// SIMATIC S7-200 project (STEP 7-Micro/WIN), CPU 221 REL 01.10

ORGANIZATION_BLOCK 主程序:OB1
TITLE=程序注释
BEGIN
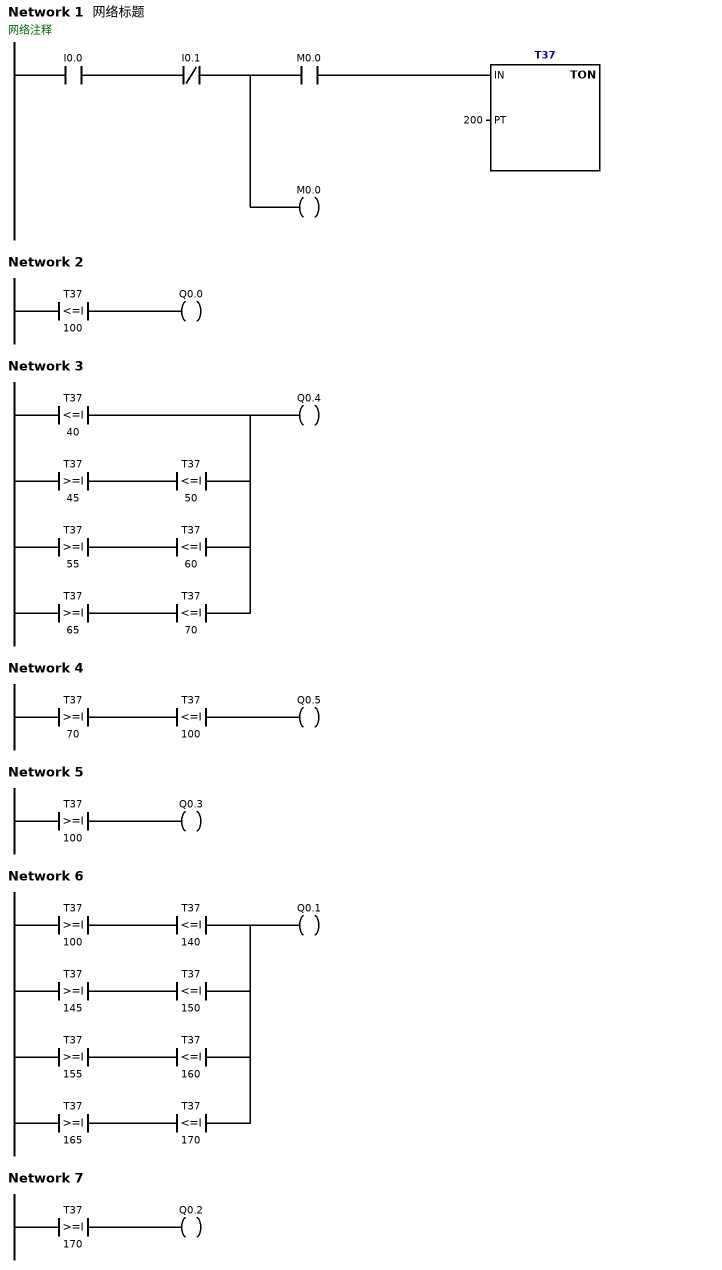
Network 1 // 网络标题
// 网络注释
LD     I0.0
AN     I0.1
LPS
A      M0.0
TON    T37, 200
LPP
=      M0.0
Network 2
LDW<=  T37, 100
=      Q0.0
Network 3
LDW<=  T37, 40
LDW>=  T37, 45
AW<=   T37, 50
OLD
LDW>=  T37, 55
AW<=   T37, 60
OLD
LDW>=  T37, 65
AW<=   T37, 70
OLD
=      Q0.4
Network 4
LDW>=  T37, 70
AW<=   T37, 100
=      Q0.5
Network 5
LDW>=  T37, 100
=      Q0.3
Network 6
LDW>=  T37, 100
AW<=   T37, 140
LDW>=  T37, 145
AW<=   T37, 150
OLD
LDW>=  T37, 155
AW<=   T37, 160
OLD
LDW>=  T37, 165
AW<=   T37, 170
OLD
=      Q0.1
Network 7
LDW>=  T37, 170
=      Q0.2
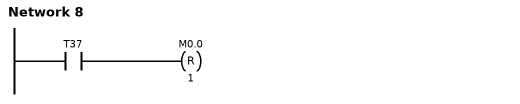
Network 8
LD     T37
R      M0.0, 1
END_ORGANIZATION_BLOCK
